{attribute 'qualified_only'}
{attribute 'strict'}
TYPE enumMode :
(
	None := 0,
	Ground := 10,
	Automat := 20,
	Manual := 30
);
END_TYPE

(* stored: Version 1.1.0.1, ProductVersion 3.1.4024.3
   DUT enumMode: Id {6c64851c-a2a6-4153-9ba4-dbc1b6cc7a1c} *)
